FUNCTION FC_CONV_M_TO_SUBPX_V2 : DINT
(*************************************************************************************************)
(*  FILENAME:    FC_CONV_M_TO_SUBPX_V2                                                           *)
(*  PROJECT:     CALMAR PUPLC                                                                    *)
(*  COPYRIGHT:   All rights reserved (c) Wifag//Polytype, Fribourg/Switzerland (2016)            *)
(*  ENVIRONMENT: TwinCAT PLC                                                                     *)
(*  VERSION:     <version>                                                                       *)
(*************************************************************************************************)
(*  DESCRIPTION:                                                                   <description> *)
(*     This function converts the value from [m] to [subpixel].                                  *)
(*                                                                                </description> *)
(*************************************************************************************************)

VAR_INPUT
  fI_Pos_M         : LREAL;             (*Position or distance in [m]*)
  fI_Res_Ph        : LREAL;             (*Printhead pixel resolution [dpi]*)
  iI_Res_SubPx     : INT;               (*Subpixel pulse resolution [pulse/px]*)
  pI_ConversionErr : POINTER TO UDINT;  (*counts catched data type conversion overflows*)
END_VAR

VAR
END_VAR

FC_CONV_M_TO_SUBPX_V2 := FC_LREAL_TO_DINT(((fI_Pos_M * 1_000_000 * fI_Res_Ph * iI_Res_SubPx) / 25400), pI_ConversionErr);

END_FUNCTION

(* stored: Version 1.1.0.1, ProductVersion 3.1.4024.9
   POU FC_CONV_M_TO_SUBPX_V2: Id {fc1692af-45c2-4eee-a342-07c4562babc7}, SpecialFunc None *)
